FUNCTION_BLOCK POSITION_MONITOR_V2 (* Composite Function Block Type *)
  (* Standard: 61499-2 *)
  (* Version 0.0, 4/30/2023, Dmitrii, Flexbridge AB, template *)
  PACKAGE UAO.Hackathon;
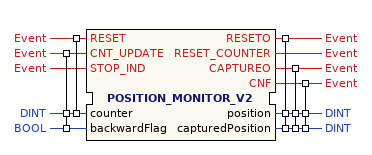
  EVENT_INPUT
    RESET WITH counter;
    CNT_UPDATE WITH counter, backwardFlag;
    STOP_IND; (* Motor stop indicatin. used to capture position *)
  END_EVENT
  EVENT_OUTPUT
    RESETO WITH position, capturedPosition; (* Reset confirmation *)
    RESET_COUNTER;
    CAPTUREO WITH position, capturedPosition; (* Position capture confirmation *)
    CNF WITH position, capturedPosition;
  END_EVENT
  VAR_INPUT
    counter : DINT;
    backwardFlag : BOOL;
  END_VAR
  VAR_OUTPUT
    position : DINT;
    capturedPosition : DINT;
  END_VAR
  FBS
    positionStorage : BASIC_STORAGE_DINT(presetValue := 0);
    FB1 : ADD_112C76C471B7A99C2; {SET_ATTRIBUTE(Configuration.GenericFBType.InterfaceParams, Runtime.Standard#CNT:=2;IN${CNT$}:DINT)}
    FB2 : SUB_112C76C471B7A99C2; {SET_ATTRIBUTE(Configuration.GenericFBType.InterfaceParams, Runtime.Standard#CNT:=2;IN${CNT$}:DINT)}
    FB3 : DS_SELECTX_158B4FD3BC4D9A1F5; {SET_ATTRIBUTE(Configuration.GenericFBType.InterfaceParams, Runtime.Standard#CNTX:=2;CNTY:=1;DI${CNTX,_,CNTY$}:DINT)}
    CaptureDelay : E_DELAY(DT := T#100ms);
    FB7 : ANY2ANY_135542315C2320DF5; {SET_ATTRIBUTE(Configuration.GenericFBType.InterfaceParams, Runtime.Standard#CNT:=1;IN${CNT$}:BOOL;OUT${CNT$}:UINT)}
    SelectOperation : E_DEMUX;
    FB4 : E_MERGE;
    FB5 : E_MERGE;
  END_FBS
  EVENT_CONNECTIONS
    RESET TO positionStorage.RESET;
    FB1.CNF TO FB3.REQ1;
    FB2.CNF TO FB3.REQ2;
    CaptureDelay.EO TO positionStorage.UPDATE;
    CNT_UPDATE TO FB7.REQ;
    FB7.CNF TO SelectOperation.EI;
    SelectOperation.EO0 TO FB1.REQ;
    SelectOperation.EO1 TO FB2.REQ;
    positionStorage.CNF TO FB4.EI1;
    FB3.IND TO FB4.EI2;
    FB4.EO TO CNF;
    positionStorage.CNF TO FB5.EI2;
    positionStorage.RESETO TO RESETO;
    positionStorage.RESETO TO FB5.EI1;
    FB5.EO TO RESET_COUNTER;
    STOP_IND TO CaptureDelay.START;
    RESET TO CaptureDelay.STOP;
    positionStorage.CNF TO CAPTUREO;
  END_CONNECTIONS
  DATA_CONNECTIONS
    positionStorage.value TO FB1.IN1;
    FB1.OUT TO FB3.DI1_1;
    positionStorage.value TO FB2.IN1;
    FB2.OUT TO FB3.DI2_1;
    FB3.OUT1 TO position;
    positionStorage.value TO capturedPosition;
    FB3.OUT1 TO positionStorage.newValue;
    FB7.OUT1 TO SelectOperation.K;
    backwardFlag TO FB7.IN1;
    counter TO FB1.IN2;
    counter TO FB2.IN2;
  END_CONNECTIONS
END_FUNCTION_BLOCK
